FUNCTION_BLOCK INTEGRATE (* Integrator with I/O for out *)
  (* Standard: 61499-1 *)
  (* Version 1.0, 2025-12-21, Franz Höpfinger, initial API and implementation and/or initial documentation *)
  PACKAGE OSCAT::Basic::POUs::Engineering::Control;
  IMPORT eclipse4diac::core::TypeHash;
  IMPORT OSCAT::Basic::POUs::Engineering::measurements::T_PLC_MS;
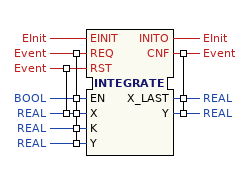
  EVENT_INPUT
    EINIT : EInit; (* Init Request *)
    REQ WITH EN, X, K, Y; (* Normal Execution Request *)
    RST WITH X; (* Reset Integrator *)
  END_EVENT
  EVENT_OUTPUT
    INITO : EInit; (* Init Confirmation *)
    CNF WITH X_LAST, Y; (* Execution Confirmation *)
  END_EVENT
  VAR_INPUT
    EN : BOOL := TRUE; (* Enable *)
    X : REAL; (* Input Value *)
    K : REAL := 1.0; (* Gain *)
  END_VAR
  VAR_OUTPUT
    X_LAST : REAL; (* Last Input Value *)
  END_VAR
  VAR_IN_OUT
    Y : REAL; (* Output Value *)
  END_VAR
  VAR
    init : BOOL := FALSE;
    last : UDINT;
    tx : UDINT;
  END_VAR
  EC_STATES
    EINIT : EINIT -> INITO;
    REQ : REQ -> CNF;
    RST : RST -> CNF;
  END_STATES
  ALGORITHM EINIT IN ST:
(* Initialization *)
init := FALSE;
  END_ALGORITHM
  ALGORITHM RST IN ST:
init := TRUE;
X_LAST := X;
  END_ALGORITHM
  ALGORITHM REQ IN ST:
(* read system time *)
tx := T_PLC_MS();

IF NOT init THEN
	this.RST();
ELSIF EN THEN
	(* Calculation: (Average X) * 1ms_in_sec * dt_ms * K + Old_Y *)
	Y := (X + X_LAST) * 0.5E-3 * UDINT_TO_REAL(tx - last) * K + Y;
	X_LAST := X;
END_IF;

last := tx;
  END_ALGORITHM
END_FUNCTION_BLOCK
